// TIA Portal V20 export
// export: Created 2025-12-01T14:57:14.9285221Z, ExportSetting None, DisplayName Totally Integrated Automation Portal, DisplayVersion V20 Update 3, DisplayName TIA Portal Openness, DisplayVersion V20 Update 3, DisplayName TIA Portal Version Control Interface, DisplayVersion V20 Update 3, DisplayName STEP 7 Professional, DisplayVersion V20 Update 3, DisplayName STEP 7 Safety, DisplayVersion V20 Update 2, DisplayName WinCC Basic/Comfort/Advanced, DisplayVersion V20 Update 3, DisplayName WinCC Professional, DisplayVersion V20 Update 3, DisplayName WinCC Unified, DisplayVersion V20 Update 3
FUNCTION_BLOCK "FB831_PasarDatosEntrePLCs_Destino"   // FB831, LAD
{ S7_Optimized_Access := 'FALSE' }
// stored: AutoNumber false, SetENOAutomatically false
   VAR_INPUT
      Mesa : UInt;
      EntrandoEnMesa : Bool;
      TransferirUT : Bool;
      In_DatosUT : Bool;
      In_Mckey_01 : "UDT_EntrePLCs";
      In_McKey_02 : "UDT_EntrePLCs";
   END_VAR
   VAR_OUTPUT
      Out_BorrarUT : Bool;
   END_VAR
   VAR
      MMcKey_01 : "UDT_EntrePLCs";
      MMckey_02 : "UDT_EntrePLCs";
      MckeyUltimo_01 : "UDT_EntrePLCs";
      MckeyUltimo_02 : "UDT_EntrePLCs";
      MemoFP_TransferirUT : Bool;
      MDatosUT : Bool;
      MBorrarUT : Bool;
   END_VAR
   VAR_TEMP
      EstadoZona : "EstadoZona";
      EstadoVI : "EstadosMesa";
      NumeroUT : UInt;
      FP_TransferirUT : Bool;
   END_VAR
   VAR_TEMP   // added for the SCL form of the ladder/FBD networks
      _w1 : Bool;
   END_VAR
BEGIN

REGION Network 1: Inicializar Variables
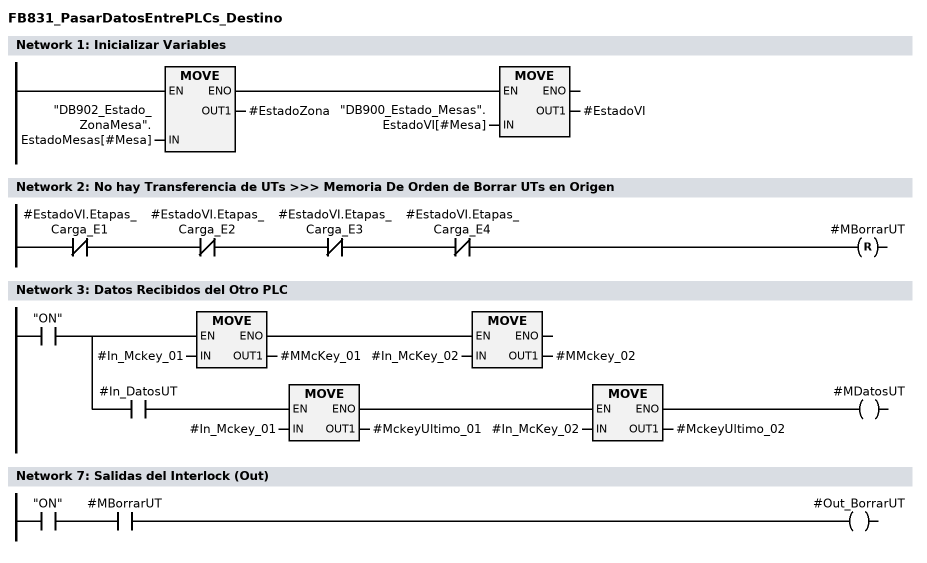
   RUNG wire#powerrail
      Move(in := "DB902_Estado_ZonaMesa".EstadoMesas[#Mesa], out1 => #EstadoZona)
      Move(in := "DB900_Estado_Mesas".EstadoVI[#Mesa], out1 => #EstadoVI)
   END_RUNG
   // the same network as SCL:
   #EstadoZona := "DB902_Estado_ZonaMesa".EstadoMesas[#Mesa];
   #EstadoVI := "DB900_Estado_Mesas".EstadoVI[#Mesa];
END_REGION

REGION Network 2: No hay Transferencia de UTs >>> Memoria De Orden de Borrar UTs en Origen
   RUNG wire#powerrail
      I_Contact( #EstadoVI.Etapas_Carga_E1 )
      I_Contact( #EstadoVI.Etapas_Carga_E2 )
      I_Contact( #EstadoVI.Etapas_Carga_E3 )
      I_Contact( #EstadoVI.Etapas_Carga_E4 )
      R_Coil( #MBorrarUT )
   END_RUNG
   // the same network as SCL:
   IF NOT #EstadoVI.Etapas_Carga_E1 AND NOT #EstadoVI.Etapas_Carga_E2 AND NOT #EstadoVI.Etapas_Carga_E3 AND NOT #EstadoVI.Etapas_Carga_E4 THEN
       #MBorrarUT := FALSE;
   END_IF;
END_REGION

REGION Network 3: Datos Recibidos del Otro PLC
   RUNG wire#powerrail
      Contact( "ON" )
      wire#w1
      Move(in := #In_Mckey_01, out1 => #MMcKey_01)
      Move(in := #In_McKey_02, out1 => #MMckey_02)
   END_RUNG
   RUNG wire#w1
      Contact( #In_DatosUT )
      Move(in := #In_Mckey_01, out1 => #MckeyUltimo_01)
      Move(in := #In_McKey_02, out1 => #MckeyUltimo_02)
      Coil( #MDatosUT )
   END_RUNG
   // the same network as SCL:
   IF "ON" THEN
       #MMcKey_01 := #In_Mckey_01;
       #MMckey_02 := #In_McKey_02;
   END_IF;
   #_w1 := "ON" AND #In_DatosUT;
   IF #_w1 THEN
       #MckeyUltimo_01 := #In_Mckey_01;
       #MckeyUltimo_02 := #In_McKey_02;
   END_IF;
   #MDatosUT := #_w1;
END_REGION

NETWORK
TITLE = Control de la Creacion de UTs entre PLCs
/////////////////////////////////////////////////////////////////////////////
/////////////////////////////////////////////////////////////////////////////
/////////////////////////////////////////////////////////////////////////////
// --- Verificacion de Orden de Transferencia de UT entre PLC's

      SET;
      A     #TransferirUT;  // Orden de Transferir la UT
      FP    #MemoFP_TransferirUT;
      =     #FP_TransferirUT;

      SET;
      AN    #FP_TransferirUT;
      JC    FinalControlUTs_EnMesa;

// --- Comprobacion Si cumple las condiciones
      SET;  // Esta Habilitado
      AN    #EntrandoEnMesa;
      JC    FinalControlUTs_EnMesa;

      SET;  // Esta Entrando Carga
      AN    #EstadoVI.Etapas_Carga_E1;
      AN    #EstadoVI.Etapas_Carga_E2;
      AN    #EstadoVI.Etapas_Carga_E3;
      AN    #EstadoVI.Etapas_Carga_E4;
      JC    FinalControlUTs_EnMesa;

/// --- Si cumple las condiciones
      JU    CrearUT_EntrePLCs;



NETWORK
TITLE = -- Creacion de UTs entre PLCs
/////////////////////////////////////////////////////////////////////////////
/////////////////////////////////////////////////////////////////////////////
/////////////////////////////////////////////////////////////////////////////
// ---    Creacion de la UT entre PLCs
// ---    * Crear UT en la Mesa con el Mckey
// ---    * Aviso de Cambio de Mesa - Codigo 11
// ---    * Y poner Destino (Normalmente la misma mesa)
CrearUT_EntrePLCs:NOP   0;
      SET;
      S     #MBorrarUT;

/////////////////////////////////////////////////////////////////////////////
// FASE 01 - Primer Mckey
      CALL  "FC721_CrearUT_EnMesa"
      ( McKey      := #In_Mckey_01.Mckey,
        MesaActual := #Mesa,
        NumeroUT   := #NumeroUT
      );

      L     11;  // Cambio de Mesa de la UT
      T     "DB812_UTs_Control".UT[#NumeroUT].EstadoEmisionUT;

      L     #In_Mckey_01.Grupo;
      T     "DB812_UTs_Control".UT[#NumeroUT].Grupo;

      L     #In_Mckey_01.TipoCarga;
      T     "DB812_UTs_Control".UT[#NumeroUT].TipoCarga;

      SET;
      A     #In_Mckey_01.AtributosDelaCarga.Vacia;
      S     "DB812_UTs_Control".UT[#NumeroUT].AtributosDelaCarga.Vacia;
      SET;
      A     #In_Mckey_01.AtributosDelaCarga.Pila;
      S     "DB812_UTs_Control".UT[#NumeroUT].AtributosDelaCarga.Pila;
      SET;
      A     #In_Mckey_01.AtributosDelaCarga.Remontada;
      S     "DB812_UTs_Control".UT[#NumeroUT].AtributosDelaCarga.Remontada;

      L     #In_Mckey_01.MesaDestino;
      T     "DB812_UTs_Control".UT[#NumeroUT].MesaDestino;
      T     "DB813_UTs_Ruta".UT[#NumeroUT].Ruta[1];
      L     #In_Mckey_01.MesaSiguienteRuta;
      T     "DB812_UTs_Control".UT[#NumeroUT].MesaIntermedia;
      T     "DB813_UTs_Ruta".UT[#NumeroUT].Ruta[0];

      SET;  // Peticion de Datos
      A     "DB850_DefinicionMesas".Mesa[#Mesa].ConfigMesa.PeticionDeDatos;
      S     "DB812_UTs_Control".UT[#NumeroUT].AtributosDeLaUT.PeticionDeDatos;


/////////////////////////////////////////////////////////////////////////////
/////////////////////////////////////////////////////////////////////////////
/////////////////////////////////////////////////////////////////////////////
// FASE 02 - Segundo Mckey
//           Mirar si hay una Segunda UT
      L     #In_McKey_02.Mckey;
      L     0;
      ==D;
      JC    FinalControlUTs_EnMesa;

/////////////////////////////////////////////////////////////////////////////
      CALL  "FC721_CrearUT_EnMesa"
      ( McKey      := #In_McKey_02.Mckey,
        MesaActual := #Mesa,
        NumeroUT   := #NumeroUT
      );

      L     11;  // Cambio de Mesa de la UT
      T     "DB812_UTs_Control".UT[#NumeroUT].EstadoEmisionUT;

      L     #In_McKey_02.Grupo;
      T     "DB812_UTs_Control".UT[#NumeroUT].Grupo;

      L     #In_McKey_02.TipoCarga;
      T     "DB812_UTs_Control".UT[#NumeroUT].TipoCarga;

      SET;
      A     #In_McKey_02.AtributosDelaCarga.Vacia;
      S     "DB812_UTs_Control".UT[#NumeroUT].AtributosDelaCarga.Vacia;
      SET;
      A     #In_McKey_02.AtributosDelaCarga.Pila;
      S     "DB812_UTs_Control".UT[#NumeroUT].AtributosDelaCarga.Pila;
      SET;
      A     #In_McKey_02.AtributosDelaCarga.Remontada;
      S     "DB812_UTs_Control".UT[#NumeroUT].AtributosDelaCarga.Remontada;

      L     #In_McKey_02.MesaDestino;
      T     "DB812_UTs_Control".UT[#NumeroUT].MesaDestino;
      T     "DB813_UTs_Ruta".UT[#NumeroUT].Ruta[1];
      L     #In_McKey_02.MesaSiguienteRuta;
      T     "DB812_UTs_Control".UT[#NumeroUT].MesaIntermedia;
      T     "DB813_UTs_Ruta".UT[#NumeroUT].Ruta[0];

      SET;  // Peticion de Datos
      A     "DB850_DefinicionMesas".Mesa[#Mesa].ConfigMesa.PeticionDeDatos;
      S     "DB812_UTs_Control".UT[#NumeroUT].AtributosDeLaUT.PeticionDeDatos;

      JU    FinalControlUTs_EnMesa;


// --- Fin de la Creacion de la UT entre PLCs
/////////////////////////////////////////////////////////////////////////////
/////////////////////////////////////////////////////////////////////////////
/////////////////////////////////////////////////////////////////////////////



NETWORK
TITLE = -- Final
/////////////////////////////////////////////////////////////////////////////
/////////////////////////////////////////////////////////////////////////////
/////////////////////////////////////////////////////////////////////////////
// --- Fin del Segmento
FinalControlUTs_EnMesa:NOP   0;



REGION Network 7: Salidas del Interlock (Out)
   RUNG wire#powerrail
      Contact( "ON" )
      Contact( #MBorrarUT )
      Coil( #Out_BorrarUT )
   END_RUNG
   // the same network as SCL:
   #Out_BorrarUT := "ON" AND #MBorrarUT;
END_REGION
END_FUNCTION_BLOCK
